Yaskawa INFORM job: turntable_cylinder_program.JBI

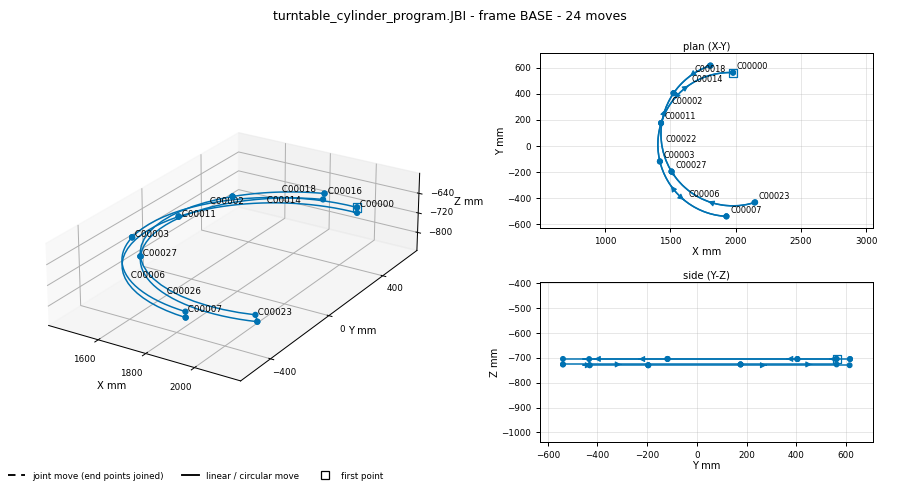
[picture p0: tool path of turntable_cylinder_program.JBI in frame BASE, 24 of 37 moves have a stored position in this frame; points joined in program order, loops and branches not executed]
/JOB
//NAME turntable_cylinder_program
//POS
///NPOS 32,0,32,0,0,0
///TOOL 0
///POSTYPE BASE
///RECTAN
///RCONF 0,0,0,0,0,0,0,0,0,0,0,0,0,0,0,0,0,0,0,0,0,0,0,0
C00000=1980.561547,562.175808,-704.153960,175.000000,-60.000000,-92.575466
C00001=1980.561547,562.175808,-704.153960,175.000000,-60.000000,-92.575466
C00002=1481.240584,291.743583,-704.153960,-175.000000,-60.000000,-30.544585
C00003=1420.272733,-118.048107,-704.153960,-175.000000,-60.000000,13.620066
C00004=1420.272733,-118.048107,-704.153960,-175.000000,-60.000000,13.620066
C00005=1420.272733,-118.048107,-704.153960,-175.000000,-60.000000,13.620066
C00006=1610.024497,-417.320678,-704.153960,-175.000000,-60.000000,51.132867
C00007=1929.574738,-538.691116,-704.153960,175.000000,-60.000000,87.271931
C00008=1930.216384,-538.721316,-726.344960,175.000000,-60.000000,87.338724
C00009=1930.216384,-538.721316,-726.344960,175.000000,-60.000000,87.338724
C00010=1544.121809,-354.553202,-726.344960,175.000000,-60.000000,41.658750
C00011=1429.791871,175.847585,-726.344960,175.000000,-60.000000,-17.330333
C00012=1429.791871,175.847585,-726.344960,175.000000,-60.000000,-17.330333
C00013=1429.791871,175.847585,-726.344960,175.000000,-60.000000,-17.330333
C00014=1632.787479,458.127043,-726.344960,-175.000000,-60.000000,-54.111752
C00015=1981.309157,562.141671,-726.344960,175.000000,-60.000000,-92.653284
C00016=1808.044087,616.303443,-704.712460,175.000000,-60.000000,-71.879883
C00017=1808.044087,616.303443,-704.712460,175.000000,-60.000000,-71.879883
C00018=1653.954897,537.242549,-704.712460,-175.000000,-60.000000,-53.796734
C00019=1525.162446,404.502760,-704.712460,-175.000000,-60.000000,-34.473853
C00020=1525.162446,404.502760,-704.712460,-175.000000,-60.000000,-34.473853
C00021=1525.162446,404.502760,-704.712460,-175.000000,-60.000000,-34.473853
C00022=1436.350000,-0.691024,-704.712460,175.000000,-60.000000,9.748099
C00023=2143.707340,-433.355857,-704.712460,175.000000,-60.000000,107.346674
C00024=2150.129766,-431.306550,-729.596460,-175.000000,-60.000000,108.047658
C00025=2150.129766,-431.306550,-729.596460,-175.000000,-60.000000,108.047658
C00026=1758.193973,-412.058950,-729.596460,175.000000,-60.000000,66.329375
C00027=1509.750575,-195.559721,-729.596460,175.000000,-60.000000,31.531356
C00028=1509.750575,-195.559721,-729.596460,175.000000,-60.000000,31.531356
C00029=1509.750575,-195.559721,-729.596460,175.000000,-60.000000,31.531356
C00030=1439.494969,202.653957,-729.596460,175.000000,-60.000000,-11.520251
C00031=1802.939975,614.605553,-729.596460,175.000000,-60.000000,-71.320559
///POSTYPE PULSE
///PULSE
EX00000=89088.0
EX00001=294912.0
///POSTYPE PULSE
///PULSE
EC00000=89088.0
EC00001=89088.0
EC00002=89088.0
EC00003=89088.0
EC00004=89088.0
EC00005=89088.0
EC00006=89088.0
EC00007=89088.0
EC00008=89088.0
EC00009=89088.0
EC00010=89088.0
EC00011=89088.0
EC00012=89088.0
EC00013=89088.0
EC00014=89088.0
EC00015=89088.0
EC00016=294912.0
EC00017=294912.0
EC00018=294912.0
EC00019=294912.0
EC00020=294912.0
EC00021=294912.0
EC00022=294912.0
EC00023=294912.0
EC00024=294912.0
EC00025=294912.0
EC00026=294912.0
EC00027=294912.0
EC00028=294912.0
EC00029=294912.0
EC00030=294912.0
EC00031=294912.0
//INST
///DATE 2023/08/16 13:45
///ATTR SC,RW,RJ
////FRAME BASE
///GROUP1 RB1,ST1
NOP
MOVJ P009 EX000 VJ=15.00
MOVJ C00000 EC00000 VJ=15.0
CALL JOB:SPYON
MOVC C00001 EC00001 V=150.0
MOVC C00002 EC00002 V=150.0
MOVC C00003 EC00003 V=150.0
MOVJ C00004 EC00004 VJ=15.0
MOVC C00005 EC00005 V=150.0
MOVC C00006 EC00006 V=150.0
MOVC C00007 EC00007 V=150.0
MOVJ C00008 EC00008 VJ=15.0
MOVC C00009 EC00009 V=150.0
MOVC C00010 EC00010 V=150.0
MOVC C00011 EC00011 V=150.0
MOVJ C00012 EC00012 VJ=15.0
MOVC C00013 EC00013 V=150.0
MOVC C00014 EC00014 V=150.0
MOVC C00015 EC00015 V=150.0
CALL JOB:SPYOF
MOVJ P009 VJ=15.00
MOVL P009 EX00000 V=150.0
MOVJ C00016 EC00016 VJ=15.0
CALL JOB:SPYON
MOVC C00017 EC00017 V=150.0
MOVC C00018 EC00018 V=150.0
MOVC C00019 EC00019 V=150.0
MOVJ C00020 EC00020 VJ=15.0
MOVC C00021 EC00021 V=150.0
MOVC C00022 EC00022 V=150.0
MOVC C00023 EC00023 V=150.0
MOVJ C00024 EC00024 VJ=15.0
MOVC C00025 EC00025 V=150.0
MOVC C00026 EC00026 V=150.0
MOVC C00027 EC00027 V=150.0
MOVJ C00028 EC00028 VJ=15.0
MOVC C00029 EC00029 V=150.0
MOVC C00030 EC00030 V=150.0
MOVC C00031 EC00031 V=150.0
CALL JOB:SPYOF
MOVJ P009 VJ=15.00
MOVL P009 EX00001 V=150.0
END
